(* CODESYS project 33_sys_module_enip_diagnostics.export

Project tree, tasks and I/O mapping:
  Device : CODESYS Control Win V3 x64, CODESYS, version 3.5.22.20
    application Application
      task ENIPScannerIOTask (cyclic, interval t#10ms, priority 0) calls EtherNet_IP_Scanner.IOCycle
      task ENIPScannerServiceTask (cyclic, interval t#20ms, priority 30) calls EtherNet_IP_Scanner.ServiceCycle
      task MainTask (cyclic, interval t#20ms, priority 1) calls PLC_PRG
      program PLC_PRG [ST]
      function block TF_Codesys_ENIP_ModuleBinding [ST]
    Ethernet : Ethernet, CODESYS, version 4.2.0.0
      EtherNet_IP_Scanner : EtherNet/IP Scanner, CODESYS, order no. 1, version 4.9.0.0
        Dev_PF525 : Generic EtherNet/IP device, CODESYS, version 4.6.0.0
            settings: INITIALIZED = TRUE; IP address of Target = [16#C0,16#A8,16#01,16#50]; Keying.Check Minor Revision = FALSE; RequiredConfigVersion = 50660864; Number of Connections = 1; Connection Settings.Requested packet interval = 10000 µs; Connection Settings.OT Connection Parameters = 18442; Connection Settings.TO Connection Parameters = 18442; Connection Settings.Connection Flags = 1056; Connection Settings.Connection Path Size = 8; Connection Settings.Large OT Connection Parameters = 1207959562; Connection Settings.Large TO Connection Parameters = 1207959562; Connection Path = [16#20,16#04,16#24,16#06,16#2C,16#02,16#2C,16#01]; Heartbeat Multiplier = 1; Input_Param0.ReadOnly = False; Input_Param0.BitSize = 8; Input_Param0.DataSize = 1; Input_Param1.ReadOnly = False; Input_Param1.BitSize = 8; Input_Param1.DataSize = 1; Input_Param2.ReadOnly = False; Input_Param2.BitSize = 8; Input_Param2.DataSize = 1; Input_Param3.ReadOnly = False; Input_Param3.BitSize = 8; Input_Param3.DataSize = 1; Input_Param4.ReadOnly = False; Input_Param4.BitSize = 8; Input_Param4.DataSize = 1; Input_Param5.ReadOnly = False; Input_Param5.BitSize = 8; Input_Param5.DataSize = 1; Input_Param6.ReadOnly = False; Input_Param6.BitSize = 8; Input_Param6.DataSize = 1; Input_Param7.ReadOnly = False; Input_Param7.BitSize = 8; Input_Param7.DataSize = 1; Output_Param0.ReadOnly = False; Output_Param0.BitSize = 8;
              Output_Param0.DataSize = 1; Output_Param1.ReadOnly = False; Output_Param1.BitSize = 8; Output_Param1.DataSize = 1; Output_Param2.ReadOnly = False; Output_Param2.BitSize = 8; Output_Param2.DataSize = 1; Output_Param3.ReadOnly = False; Output_Param3.BitSize = 8; Output_Param3.DataSize = 1; Input_Param0.Name = 'Input_Param0'; Input_Param0.HelpString = ''; Input_Param0.ReadOnly = False; Input_Param0.BitSize = 8; Input_Param0.DataSize = 1; Input_Param0.DataType = 'BYTE'; Input_Param1.Name = 'Input_Param1'; Input_Param1.HelpString = ''; Input_Param1.ReadOnly = False; Input_Param1.BitSize = 8; Input_Param1.DataSize = 1; Input_Param1.DataType = 'BYTE'; Input_Param2.Name = 'Input_Param2'; Input_Param2.HelpString = ''; Input_Param2.ReadOnly = False; Input_Param2.BitSize = 8; Input_Param2.DataSize = 1; Input_Param2.DataType = 'BYTE'; Input_Param3.Name = 'Input_Param3'; Input_Param3.HelpString = ''; Input_Param3.ReadOnly = False; Input_Param3.BitSize = 8; Input_Param3.DataSize = 1; Input_Param3.DataType = 'BYTE'; Input_Param4.Name = 'Input_Param4'; Input_Param4.HelpString = ''; Input_Param4.ReadOnly = False; Input_Param4.BitSize = 8; Input_Param4.DataSize = 1; Input_Param4.DataType = 'BYTE';
              Input_Param5.Name = 'Input_Param5'; Input_Param5.HelpString = ''; Input_Param5.ReadOnly = False; Input_Param5.BitSize = 8; Input_Param5.DataSize = 1; Input_Param5.DataType = 'BYTE'; Input_Param6.Name = 'Input_Param6'; Input_Param6.HelpString = ''; Input_Param6.ReadOnly = False; Input_Param6.BitSize = 8; Input_Param6.DataSize = 1; Input_Param6.DataType = 'BYTE'; Input_Param7.Name = 'Input_Param7'; Input_Param7.HelpString = ''; Input_Param7.ReadOnly = False; Input_Param7.BitSize = 8; Input_Param7.DataSize = 1; Input_Param7.DataType = 'BYTE'; Output_Param0.Name = 'Output_Param0'; Output_Param0.HelpString = ''; Output_Param0.ReadOnly = False; Output_Param0.BitSize = 8; Output_Param0.DataSize = 1; Output_Param0.DataType = 'BYTE'; Output_Param1.Name = 'Output_Param1'; Output_Param1.HelpString = ''; Output_Param1.ReadOnly = False; Output_Param1.BitSize = 8; Output_Param1.DataSize = 1; Output_Param1.DataType = 'BYTE'; Output_Param2.Name = 'Output_Param2'; Output_Param2.HelpString = ''; Output_Param2.ReadOnly = False; Output_Param2.BitSize = 8; Output_Param2.DataSize = 1; Output_Param2.DataType = 'BYTE'; Output_Param3.Name = 'Output_Param3'; Output_Param3.HelpString = ''; Output_Param3.ReadOnly = False; Output_Param3.BitSize = 8;
              Output_Param3.DataSize = 1; Output_Param3.DataType = 'BYTE'; ConfigVersion = 50660864
            unmapped channels: Input_Param0, Input_Param1, Input_Param2, Input_Param3, Input_Param4, Input_Param5, Input_Param6, Input_Param7, Output_Param0, Output_Param1, Output_Param2, Output_Param3
*)

// Device/Application/PLC_PRG
PROGRAM PLC_PRG
VAR
	fbModuleBinding: TF_Codesys_ENIP_ModuleBinding;
	fbReconfigure : DED.Reconfigure;
	
	xInp_Inhibit : BOOL;
	xInp_Uninhibit : BOOL;
	
	xInp_Connected: BOOL;
	xInp_Enabled: BOOL;
	xInp_Faulted: BOOL;
	xInp_DiagnosticAvailable: BOOL;
	xInp_CanReconfigure: BOOL;
	xInp_ReconfigureBusy: BOOL;
	xInp_ReconfigureDone: BOOL;
	xInp_ReconfigureFailed: BOOL;
	xOut_Connected: BOOL;
	xOut_Enabled: BOOL;
	xOut_Faulted: BOOL;
	xOut_DiagnosticAvailable: BOOL;
	xOut_RequestReconfigure: BOOL;
	xOut_RequestedEnable: BOOL;
	xOut_ReconfigureBlocked: BOOL;
	xOut_ReconfigureBusy: BOOL;
	xOut_ReconfigureDone: BOOL;
	xOut_ReconfigureFailed: BOOL;
	xObservedEnabled : BOOL;
	xObservedDiagnosticAvailable : BOOL;
	sObservedDiagnostic : STRING(255);
	eObservedDeviceState : DED.DEVICE_STATE;
	eObservedReconfigureError : DED.ERROR;
END_VAR

xObservedEnabled := Dev_PF525.Enable;
xObservedDiagnosticAvailable := Dev_PF525.xDiagnosticAvailable;
sObservedDiagnostic := Dev_PF525.sDiagString;
eObservedDeviceState := Dev_PF525.GetDeviceState();

xInp_CanReconfigure :=
    DED.CanReconfigure(itfNode := Dev_PF525);
    
xInp_Connected :=
    (Dev_PF525.eState = IoDrvEtherNetIP.AdapterState.RUNNING)
    AND
    (eObservedDeviceState = DED.DEVICE_STATE.RUNNING);

xInp_Enabled := Dev_PF525.Enable;

xInp_Faulted :=
    (Dev_PF525.eState = IoDrvEtherNetIP.AdapterState.BUS_ERROR)
    OR
	(Dev_PF525.eState = IoDrvEtherNetIP.AdapterState.ERROR)
    OR
    (eObservedDeviceState = DED.DEVICE_STATE.ERROR);

xInp_DiagnosticAvailable :=
    Dev_PF525.xDiagnosticAvailable;
	
xInp_ReconfigureBusy :=
    fbReconfigure.xBusy;

xInp_ReconfigureDone :=
    fbReconfigure.xDone;

xInp_ReconfigureFailed :=
    fbReconfigure.xError;

eObservedReconfigureError :=
    fbReconfigure.eError;

fbModuleBinding(
    Inp_Connected := xInp_Connected,
    Inp_Enabled := xInp_Enabled,
    Inp_Faulted := xInp_Faulted,
    Inp_DiagnosticAvailable := xInp_DiagnosticAvailable,
    Inp_CanReconfigure := xInp_CanReconfigure,
    Inp_ReconfigureBusy := xInp_ReconfigureBusy,
    Inp_ReconfigureDone := xInp_ReconfigureDone,
    Inp_ReconfigureFailed := xInp_ReconfigureFailed,
    Inp_Inhibit := xInp_Inhibit,
    Inp_Uninhibit := xInp_Uninhibit,
    Out_Connected => xOut_Connected,
    Out_Enabled => xOut_Enabled,
    Out_Faulted => xOut_Faulted,
    Out_DiagnosticAvailable => xOut_DiagnosticAvailable,
    Out_RequestReconfigure => xOut_RequestReconfigure,
    Out_RequestedEnable => xOut_RequestedEnable,
    Out_ReconfigureBlocked => xOut_ReconfigureBlocked,
    Out_ReconfigureBusy => xOut_ReconfigureBusy,
    Out_ReconfigureDone => xOut_ReconfigureDone,
    Out_ReconfigureFailed => xOut_ReconfigureFailed
);

IF xOut_RequestReconfigure THEN
    Dev_PF525.Enable := xOut_RequestedEnable;
END_IF;

fbReconfigure(
    xExecute := xOut_RequestReconfigure,
    itfNode := Dev_PF525
);

END_PROGRAM

// Device/Application/TF_Codesys_ENIP_ModuleBinding
FUNCTION_BLOCK TF_Codesys_ENIP_ModuleBinding
VAR_INPUT
	Inp_Connected: BOOL;
	Inp_Enabled: BOOL;
	Inp_Faulted: BOOL;
	Inp_DiagnosticAvailable: BOOL;
	Inp_CanReconfigure: BOOL;
	Inp_ReconfigureBusy: BOOL;
	Inp_ReconfigureDone: BOOL;
	Inp_ReconfigureFailed: BOOL;
	Inp_Inhibit: BOOL;
	Inp_Uninhibit: BOOL;
END_VAR
VAR_OUTPUT
	Out_Connected: BOOL;
	Out_Enabled: BOOL;
	Out_Faulted: BOOL;
	Out_DiagnosticAvailable: BOOL;
	Out_RequestReconfigure: BOOL;
	Out_RequestedEnable: BOOL;
	Out_ReconfigureBlocked: BOOL;
	Out_ReconfigureBusy: BOOL;
	Out_ReconfigureDone: BOOL;
	Out_ReconfigureFailed: BOOL;
END_VAR
VAR
	CommandLatch: BOOL;
END_VAR

Out_Connected := Inp_Connected;
Out_Enabled := Inp_Enabled;
Out_Faulted := Inp_Faulted;
Out_DiagnosticAvailable := Inp_DiagnosticAvailable;
Out_ReconfigureBusy := Inp_ReconfigureBusy;
Out_ReconfigureDone := Inp_ReconfigureDone;
Out_ReconfigureFailed := Inp_ReconfigureFailed;
Out_RequestReconfigure := FALSE;
IF ((Inp_Inhibit OR Inp_Uninhibit) AND NOT (CommandLatch)) THEN
    IF (Inp_CanReconfigure AND NOT (Inp_ReconfigureBusy)) THEN
        Out_RequestedEnable := NOT (Inp_Inhibit);
        Out_RequestReconfigure := TRUE;
        Out_ReconfigureBlocked := FALSE;
    ELSE
        Out_ReconfigureBlocked := TRUE;
    END_IF;
END_IF;
IF Inp_ReconfigureDone THEN
    Out_ReconfigureBlocked := FALSE;
END_IF;
CommandLatch := (Inp_Inhibit OR Inp_Uninhibit);

END_FUNCTION_BLOCK
